TYPE Status_Typ :
STRUCT
	SessionCounter:UINT;
END_STRUCT
END_TYPE

(* stored: Version 1.1.0.1, ProductVersion 3.1.4024.3
   DUT Status_Typ: Id {d3f865a8-88db-4823-a365-8f3c93512b7b} *)
